Fanuc KAREL source: ka00001.KL

PROGRAM KA00001
%NOLOCKGROUP
VAR
SRC:INTEGER;DST:INTEGER
BEGIN
--
SRC=2
DST=SRC
END KA00001
